// TIA Portal V16 export
// export: Created 2021-11-12T13:31:04.0098191Z, ExportSetting WithDefaults, DisplayName Totally Integrated Automation Portal, DisplayVersion V16 Update 3, DisplayName TIA Portal Version Control Interface, DisplayVersion V16 Update 2, DisplayName TIA Portal Openness, DisplayVersion V16 Update 3, DisplayName SINAMICS Startdrive Advanced, DisplayVersion V16 Update 5, DisplayName SINAMICS Startdrive G130, G150, S120, S150, SINAMICS MV, S210, DisplayVersion V16 Update 5, DisplayName SINAMICS Startdrive G110M, G120, G120C, G120D, G120P, G115D, DisplayVersion V16 Update 5, DisplayName STEP 7 Professional, DisplayVersion V16 Update 3, DisplayName STEP 7 Safety, DisplayVersion V16, DisplayName WinCC UA Professional, DisplayVersion V16 Update 3
DATA_BLOCK "IDB_DataColl"   // DB195
{ DB_Accessible_From_OPC_UA := 'FALSE' }
VERSION : 0.1
// stored: AutoNumber true, DBAccessibleFromOPCUA false, InstanceOfName DataColl, InstanceOfType FB
"DataColl"
   // VAR
   //    SS_Edge : Array[0..9] of Bool;
   //    SF_ArchivePeriodicallyFullAlarm : "STD_DI_Mon";
   //    SF_ArchivePeriodicallyFullWarn : "STD_DI_Mon";
   //    SF_ArchiveItemFullAlarm : "STD_DI_Mon";
   //    SF_ArchiveItemFullWarn : "STD_DI_Mon";
   //    SF_FIFOQueueArchivePeriodically : "FIFOQueueArchivPeriodically";
   //    SF_FIFOQueueArchiveItem : "FIFOQueueArchivItem";
   //    SI_PointerArchivePeriodically : Int;
   //    SI_PointerArchiveItem : Int;
   //    SB1_BufferArchivePeriodicallyFullAlarm : Bool;
   //    SB1_BufferArchivePeriodicallyFullWarn : Bool;
   //    SB1_BufferArchiveItemFullAlarm : Bool;
   //    SB1_BufferArchiveItemFullWarn : Bool;
   // END_VAR
BEGIN
END_DATA_BLOCK
